(*********************************** G.D S.p.A. - Technical Department ***********************************
============= PROGRAM INFO ============
FOLDER:             TBD
MACHINES INVOLVED:  TBD 

============= DESCRIPTION =============
csp main interface program

============= REVISIONS ===============
Date		Version	 	Author      	Description             
----------	-------		------------  	--------------------------------------------
2019/09/27 	0000.00	 	M.Grasso		Creation of the PRG

**********************************************************************************************************)
PROGRAM _csp_case_loader_highest
VAR
END_VAR

csp_case_loader();

(* CASE *)
	(* LOADER *)
		(* PUSHER *)
		csp_case_loader_pusher();
		(* SENSORS *)
		csp_case_loader_virtualMaster();

END_PROGRAM

(* stored: Version 1.1.0.1, ProductVersion 3.1.4024.3
   POU _csp_case_loader_highest: Id {14c76e5c-f3c2-4c8d-9773-8e8ca780976f}, SpecialFunc None *)
